TYPE ST_TCEvents :
STRUCT
	arrTCEvents : ARRAY [1..10]  OF ST_Event;
	
END_STRUCT
END_TYPE

(* stored: Version 1.1.0.1, ProductVersion 3.1.4022.10
   DUT ST_TCEvents: Id {401815fb-7821-4902-a63e-c14d0a0cf325} *)
